// TIA Portal V21 export
FUNCTION "LINEAR" : Void   // FC15, LAD
{ S7_Optimized_Access := 'TRUE' }
// stored: SetENOAutomatically false
   VAR_INPUT
      "ENGG MIN" : Int;
      "ENGG MAX" : Int;
      "SCL MIN" : Real;
      "SCL MAX" : Real;
      AI : Int;
   END_VAR
   VAR_OUTPUT
      ACTUAL : Real;
   END_VAR
   VAR_TEMP
      NOM : Real;
   END_VAR
BEGIN

REGION Network 1
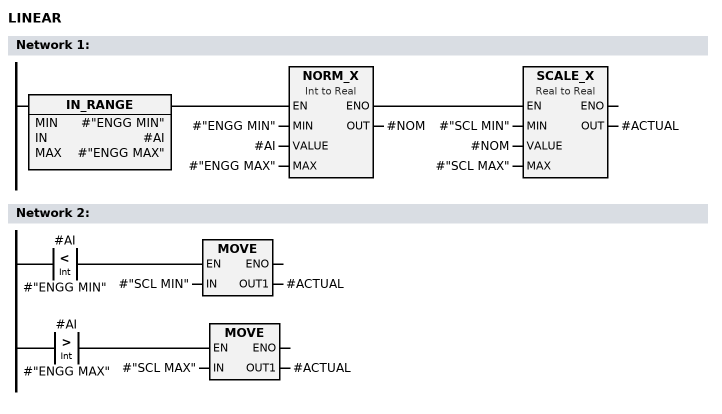
   RUNG wire#powerrail
      { S7_Templates := "SrcType := Int" } InRange(min := #"ENGG MIN", in := #AI, max := #"ENGG MAX")
      { S7_Templates := "[SrcType := Int, DestType := Real]" } Normalize(min := #"ENGG MIN", value := #AI, max := #"ENGG MAX", out => #NOM)
      { S7_Templates := "[SrcType := Real, DestType := Real]" } Scale(min := #"SCL MIN", value := #NOM, max := #"SCL MAX", out => #ACTUAL)
   END_RUNG
   // the same network as SCL:
   IF (#"ENGG MIN" <= #AI) AND (#AI <= #"ENGG MAX") THEN
       #NOM := NORM_X(MIN := #"ENGG MIN", VALUE := #AI, MAX := #"ENGG MAX");
       #ACTUAL := SCALE_X(MIN := #"SCL MIN", VALUE := #NOM, MAX := #"SCL MAX");
   END_IF;
END_REGION

REGION Network 2
   RUNG wire#powerrail
      { S7_Templates := "SrcType := Int" } LT_Contact(in1 := #AI, in2 := #"ENGG MIN")
      Move(in := #"SCL MIN", out1 => #ACTUAL)
   END_RUNG
   RUNG wire#powerrail
      { S7_Templates := "SrcType := Int" } GT_Contact(in1 := #AI, in2 := #"ENGG MAX")
      Move(in := #"SCL MAX", out1 => #ACTUAL)
   END_RUNG
   // the same network as SCL:
   IF #AI < #"ENGG MIN" THEN #ACTUAL := #"SCL MIN"; END_IF;
   IF #AI > #"ENGG MAX" THEN #ACTUAL := #"SCL MAX"; END_IF;
END_REGION
END_FUNCTION
